{attribute 'c++_compatible'}
FUNCTION_BLOCK FB_ConditionMoreThanFive IMPLEMENTS ITcVnCustomElementCondition_ITcVnContainer
VAR_INPUT
END_VAR
VAR_OUTPUT
END_VAR
VAR
END_VAR

{attribute 'c++_compatible'}
{attribute 'minimal_input_size' := '4'}
{attribute 'pack_mode' := '4'}
(* Evaluates the condition for the container. *)
METHOD Condition : BOOL
VAR_INPUT
	ipElement			:	ITcVnContainer;
END_VAR
VAR
	nNumberOfElements	:	ULINT;
	hr					:	HRESULT;
END_VAR
hr := F_VN_GetNumberOfElements(ipElement, nNumberOfElements, hr);
IF FAILED(hr) OR nNumberOfElements <= 5 THEN
	Condition := FALSE;
ELSE
	Condition := TRUE;
END_IF
END_METHOD

END_FUNCTION_BLOCK

(* stored: Version 1.1.0.1, ProductVersion 3.1.4024.3
   POU FB_ConditionMoreThanFive: Id {ba18a29d-0000-4bc7-b79a-75246b9e15fc}, SpecialFunc None
   Method Condition: Id {2eb2806b-612b-4868-8e00-1de8edaf61bc} *)
